// TIA Portal V16 export
// export: Created 2024-12-03T15:41:44.8002036Z, ExportSetting WithReadOnly, DisplayName Totally Integrated Automation Portal, DisplayVersion V16 Update 6, DisplayName TIA Portal Version Control Interface, DisplayVersion V16 Update 2, DisplayName TIA Portal Openness, DisplayVersion V16 Update 6, DisplayName TIA Portal Teamcenter Gateway, DisplayVersion V16, DisplayName SINAMICS Startdrive Advanced, DisplayVersion V16 Update 5, DisplayName SINAMICS Startdrive G130, G150, S120, S150, SINAMICS MV, S210, DisplayVersion V16 Update 5, DisplayName SINAMICS Startdrive G110M, G120, G120C, G120D, G120P, G115D, DisplayVersion V16 Update 5, DisplayName STEP 7 Professional, DisplayVersion V16 Update 6, DisplayName STEP 7 Safety, DisplayVersion V16, DisplayName WinCC Advanced / Unified PC, DisplayVersion V16 Update 6
TYPE "typeDiagnostics"
TITLE = typeDiagnostics
// Provides a structure for detailed diagnostics
// stored: CreationDate 2022-04-18T07:33:35.9561163Z, InterfaceModifiedDate 2022-04-18T07:33:44.4399127Z, IsConsistent true, LibraryConformanceStatus The object is library-conformant., ModifiedDate 2022-04-18T07:33:44.4399127Z
   STRUCT
      status { ExternalVisible := 'False'; ExternalWritable := 'False'} : Word;   // Status of the block or error identification when error occurred
      subfunctionStatus { ExternalVisible := 'False'; ExternalWritable := 'False'} : DWord;   // Status or return value of called FBs, FCs and system blocks
      stateNumber { ExternalVisible := 'False'; ExternalWritable := 'False'} : DInt;   // State in the state machine of the block where the error occurred
   END_STRUCT;
END_TYPE
